Universal Robots PolyScope program: polyscope.in.memory.program.urp

Program <unnamed> (installation=default directory=/programs createdIn=5.9.5.1031259 lastSavedIn=5.9.5.1031259 robotSerialNumber=20195500451)
Robot Program (runOnlyOnce=false)
  Placeholder
